# EPICS substitutions: ek9000App/Db/EL1808.substitutions
file EL1808.template
{ 	pattern
	{
		TERMINAL,

	}
	{
	}
}
